(* IEC 61131-3 sources: com.logicals.lc3.webinar/usRTS_RPMControl_iSOC/src_FB_LIB_SAFE/Safe/Numeric, 4 files *)

(* ---- wADD_SAFEINT.iecst ---- *)
NAMESPACE logicals.web.standard.safe
NAMESPACE numeric

/*
 * Function block wrapper for IEC 61131-3 ADD<br>
 * IN1 =  1st value (SAFEINT)<br>
 * IN2 =  2nd value (SAFEINT)<br>
 * OUT = Sum of all input values (SAFEINT)<br>
 */
FUNCTION_BLOCK wADD_SAFEINT
	{ vNameAlignment:="center"; altName:="+"; bgColor:="GoldenRod"; width:=40; hideIONames; }
	VAR_INPUT
		IN1 : SAFEINT;
		IN2 : SAFEINT;
	END_VAR
	VAR_OUTPUT
		OUT : SAFEINT;
	END_VAR

	OUT := ADD(IN1:=IN1, IN2:=IN2, ENO=>ENO);
END_FUNCTION_BLOCK

END_NAMESPACE
END_NAMESPACE

(* ---- wDIV_SAFEINT.iecst ---- *)
NAMESPACE logicals.web.standard.safe
NAMESPACE numeric

/*
 * Function block wrapper for IEC 61131-3 DIV<br>
 * IN1 =  1st value (SAFEINT)<br>
 * IN2 =  2nd value (SAFEINT)<br>
 * OUT = Quotient of IN1 divided by IN2 (SAFEINT)<br>
 */
FUNCTION_BLOCK wDIV_SAFEINT
	{ vNameAlignment:="center"; altName:="/"; bgColor:="GoldenRod"; width:=40; hideIONames; }
	VAR_INPUT
		IN1 : SAFEINT;
		IN2 : SAFEINT;
	END_VAR
	VAR_OUTPUT
		OUT : SAFEINT;
	END_VAR

	OUT := DIV(IN1:=IN1, IN2:=IN2, ENO=>ENO);
END_FUNCTION_BLOCK

END_NAMESPACE
END_NAMESPACE

(* ---- wMUL_SAFEINT.iecst ---- *)
NAMESPACE logicals.web.standard.safe
NAMESPACE numeric

/*
 * Function block wrapper for IEC 61131-3 MUL<br>
 * IN1 =  1st value (SAFEINT)<br>
 * IN2 =  2nd value (SAFEINT)<br>
 * OUT = Product of multiplication of all inputs (SAFEINT)<br>
 */
FUNCTION_BLOCK wMUL_SAFEINT
	{ vNameAlignment:="center"; altName:="*"; bgColor:="GoldenRod"; width:=40; hideIONames; }
	VAR_INPUT
		IN1 : SAFEINT;
		IN2 : SAFEINT;
	END_VAR
	VAR_OUTPUT
		OUT : SAFEINT;
	END_VAR

	OUT := MUL(IN1:=IN1, IN2:=IN2, ENO=>ENO);
END_FUNCTION_BLOCK

END_NAMESPACE
END_NAMESPACE

(* ---- wSUB_SAFEINT.iecst ---- *)
NAMESPACE logicals.web.standard.safe
NAMESPACE numeric

/*
 * Function block wrapper for IEC 61131-3 SUB<br>
 * IN1 =  1st value (SAFEINT)<br>
 * IN2 =  2nd value (SAFEINT)<br>
 * OUT = IN1 minus IN2 (SAFEINT)<br>
 */
FUNCTION_BLOCK wSUB_SAFEINT
	{ vNameAlignment:="center"; altName:="-"; bgColor:="GoldenRod"; width:=40; hideIONames; }
	VAR_INPUT
		IN1 : SAFEINT;
		IN2 : SAFEINT;
	END_VAR
	VAR_OUTPUT
		OUT : SAFEINT;
	END_VAR

	OUT := SUB(IN1:=IN1, IN2:=IN2, ENO=>ENO);
END_FUNCTION_BLOCK

END_NAMESPACE
END_NAMESPACE
